// Template of event classes.
FUNCTION_BLOCK FB_BA_EC01 EXTENDS FB_BA_View
VAR CONSTANT
	OBJECT_NAME			: STRING					:= 'EC{InstID}';
END_VAR
VAR
	{region 'Alarm'}
		AlmSmpl			: FB_BA_EC := (
							iParent					:= THIS^,
							nInstanceID				:= MyECIDs.AlmSmpl,
							sObjectName				:= OBJECT_NAME,
							sDescription			:= '{Alarm (Einfach)}',
							eEventType				:= E_BA_EventType.eAlarm,
							eAlarmMode				:= E_BA_AlarmMode.eSimple,
							aPriority				:= [ 10, 11, 12 ]
						);
		AlmStd			: FB_BA_EC := (
							iParent					:= THIS^,
							nInstanceID				:= MyECIDs.AlmStd,
							sObjectName				:= OBJECT_NAME,
							sDescription			:= '{Alarm (Standard)}',
							eEventType				:= E_BA_EventType.eAlarm,
							eAlarmMode				:= E_BA_AlarmMode.eStandard,
							aPriority				:= [ 13, 14, 15 ]
						);
		AlmExt			: FB_BA_EC := (
							iParent					:= THIS^,
							nInstanceID				:= MyECIDs.AlmExt,
							sObjectName				:= OBJECT_NAME,
							sDescription			:= '{Alarm (Erweitert)}',
							eEventType				:= E_BA_EventType.eAlarm,
							eAlarmMode				:= E_BA_AlarmMode.eExtended,
							aPriority				:= [ 16, 17, 18 ]
						);
	{endregion}
	{region 'Disturb'}
		DstSmpl			: FB_BA_EC	:= (
							iParent					:= THIS^,
							nInstanceID				:= MyECIDs.DstSmpl,
							sObjectName				:= OBJECT_NAME,
							sDescription			:= '{Störung (Einfach)}',
							eEventType				:= E_BA_EventType.eDisturb,
							eAlarmMode				:= E_BA_AlarmMode.eSimple,
							aPriority				:= [ 50, 51, 52 ]
						);
		DstStd			: FB_BA_EC := (
							iParent					:= THIS^,
							nInstanceID				:= MyECIDs.DstStd,
							sObjectName				:= OBJECT_NAME,
							sDescription			:= '{Störung (Standard)}',
							eEventType				:= E_BA_EventType.eDisturb,
							eAlarmMode				:= E_BA_AlarmMode.eStandard,
							aPriority				:= [ 53, 54, 55 ]
						);
		DstExt			: FB_BA_EC := (
							iParent					:= THIS^,
							nInstanceID				:= MyECIDs.DstExt,
							sObjectName				:= OBJECT_NAME,
							sDescription			:= '{Störung (Erweitert)}',
							eEventType				:= E_BA_EventType.eDisturb,
							eAlarmMode				:= E_BA_AlarmMode.eExtended,
							aPriority				:= [ 56, 57, 58 ]
						);
	{endregion}
	{region 'Maintenance'}
		MntnSmpl		: FB_BA_EC := (
							iParent					:= THIS^,
							nInstanceID				:= MyECIDs.MntnSmpl,
							sObjectName				:= OBJECT_NAME,
							sDescription			:= '{Wartung (Einfach)}',
							eEventType				:= E_BA_EventType.eMaintenance,
							eAlarmMode				:= E_BA_AlarmMode.eSimple,
							aPriority				:= [ 90, 91, 92 ]
						);
		MntnStd			: FB_BA_EC := (
							iParent					:= THIS^,
							nInstanceID				:= MyECIDs.MntnStd,
							sObjectName				:= OBJECT_NAME,
							sDescription			:= '{Wartung (Standard)}',
							eEventType				:= E_BA_EventType.eMaintenance,
							eAlarmMode				:= E_BA_AlarmMode.eStandard,
							aPriority				:= [ 93, 94, 95 ]
						);

		MntnExt			: FB_BA_EC := (
							iParent					:= THIS^,
							nInstanceID				:= MyECIDs.MntnExt,
							sObjectName				:= OBJECT_NAME,
							sDescription			:= '{Wartung (Erweitert)}',
							eEventType				:= E_BA_EventType.eMaintenance,
							eAlarmMode				:= E_BA_AlarmMode.eExtended,
							aPriority				:= [ 96, 97, 98 ]
						);
	{endregion}
	{region 'Notification'}
		NtfSmpl			: FB_BA_EC := (
							iParent					:= THIS^,
							nInstanceID				:= MyECIDs.NtfSmpl,
							sObjectName				:= OBJECT_NAME,
							sDescription			:= '{Benachrichtigung (Einfach)}',
							eEventType				:= E_BA_EventType.eNotification,
							eAlarmMode				:= E_BA_AlarmMode.eSimple,
							aPriority				:= [ 130, 131, 132 ]
						);
		NtfStd			: FB_BA_EC := (
							iParent					:= THIS^,
							nInstanceID				:= MyECIDs.NtfStd,
							sObjectName				:= OBJECT_NAME,
							sDescription			:= '{Benachrichtigung (Standard)}',
							eEventType				:= E_BA_EventType.eNotification,
							eAlarmMode				:= E_BA_AlarmMode.eStandard,
							aPriority				:= [ 133, 134, 135 ]
						);
	{endregion}
	{region 'Other'}
		OthSmpl			: FB_BA_EC := (
							iParent					:= THIS^,
							nInstanceID				:= MyECIDs.OthSmpl,
							sObjectName				:= OBJECT_NAME,
							sDescription			:= '{Sonstiges (Einfach)}',
							eEventType				:= E_BA_EventType.eOther,
							eAlarmMode				:= E_BA_AlarmMode.eSimple,
							aPriority				:= [ 180, 181, 182 ]
						);
		OthStd			: FB_BA_EC := (
							iParent					:= THIS^,
							nInstanceID				:= MyECIDs.OthStd,
							sObjectName				:= OBJECT_NAME,
							sDescription			:= '{Sonstiges (Standard)}',
							eEventType				:= E_BA_EventType.eOther,
							eAlarmMode				:= E_BA_AlarmMode.eStandard,
							aPriority				:= [ 183, 184, 185 ]
						);
	{endregion}
END_VAR

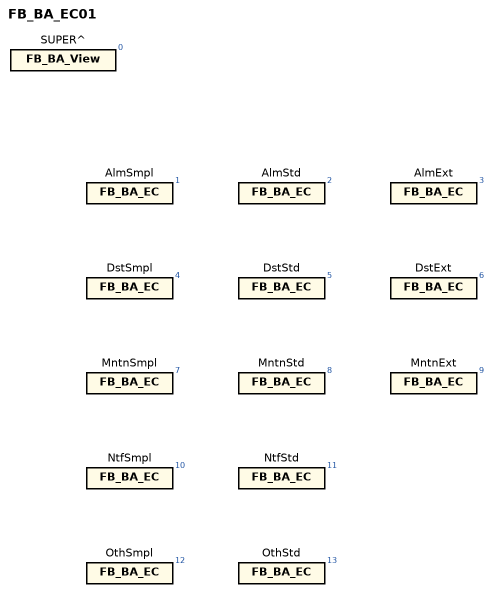
SUPER^(); // FB_BA_View
AlmSmpl(); // FB_BA_EC
AlmStd(); // FB_BA_EC
AlmExt(); // FB_BA_EC
DstSmpl(); // FB_BA_EC
DstStd(); // FB_BA_EC
DstExt(); // FB_BA_EC
MntnSmpl(); // FB_BA_EC
MntnStd(); // FB_BA_EC
MntnExt(); // FB_BA_EC
NtfSmpl(); // FB_BA_EC
NtfStd(); // FB_BA_EC
OthSmpl(); // FB_BA_EC
OthStd(); // FB_BA_EC

END_FUNCTION_BLOCK

(* stored: Version 1.1.0.1, ProductVersion 3.1.4024.12
   POU FB_BA_EC01: Id {4e92d919-3d0a-42aa-8547-5b7fc4caebbe}, SpecialFunc None *)
